FUNCTION_BLOCK F_LT (* equality *)
  (* Standard: 61131-3; Classification: standard comparison function *)
  (* Version 1.0, 2011-09-29, 4DIAC-IDE, 4DIAC-Consortium *)
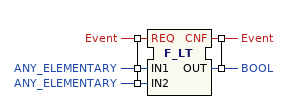
  EVENT_INPUT
    REQ WITH IN1, IN2; (* Service Request *)
  END_EVENT
  EVENT_OUTPUT
    CNF WITH OUT; (* Confirmation of Requested Service *)
  END_EVENT
  VAR_INPUT
    IN1 : ANY_ELEMENTARY; (* Input value 1 *)
    IN2 : ANY_ELEMENTARY; (* Input value 2 *)
  END_VAR
  VAR_OUTPUT
    OUT : BOOL; (* value 1 < value2 = true *)
  END_VAR
END_FUNCTION_BLOCK
